% RSLogix 500 project pid_driving_pwm_analog_servo_sine_0.5-2.5ms.RSS, saved by version 8.30.00.16 %
PROJECT "UNTITLED"    % processor: Bul.1763 MicroLogix 1100 Series B %

PROGRAM FILES
  LAD 2 "CONTINUOUS"  7 rungs
  LAD 3 "DRIVESERVO"  3 rungs
  LAD 4 "PID_SCHED"  7 rungs
  LAD 5 "SINE_SIMUL"  7 rungs

DATA FILES
  O0 OUTPUT  4 elements
  I1 INPUT  6 elements
  S2 STATUS  66 elements
  B3 BINARY  1 elements
  T4 TIMER  1 elements
  C5 COUNTER  1 elements
  R6 CONTROL  1 elements
  N7 INTEGER  30 elements
  F8 FLOAT  4 elements
  L9 LONGS  8 elements
  PD10   1 elements

LADDER 2 "CONTINUOUS"
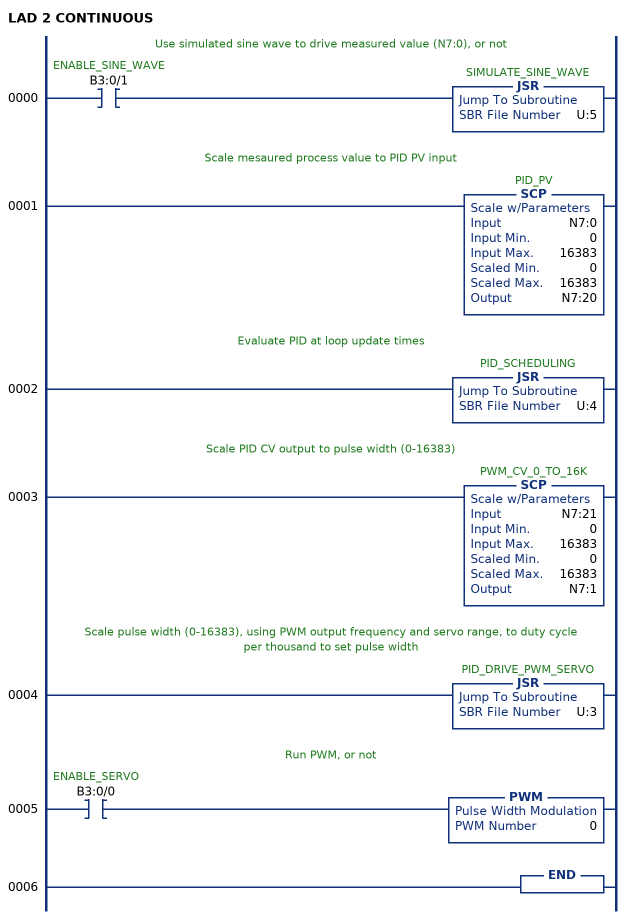
% Rung: 0 %
% Use simulated sine wave to drive measured value (N7:0), or not %
SOR XIC B3:0/1 JSR U:5 EOR
%   B3:0/1  ENABLE_SINE_WAVE %
%   U:5  SIMULATE_SINE_WAVE %
% Rung: 1 %
% Scale mesaured process value to PID PV input %
SOR SCP N7:0 0 16383 0 16383 N7:20 EOR
%   N7:0  MEASURED_VALUE %
%   N7:20  PID_PV %
% Rung: 2 %
% Evaluate PID at loop update times %
SOR JSR U:4 EOR
%   U:4  PID_SCHEDULING %
% Rung: 3 %
% Scale PID CV output to pulse width (0-16383) %
SOR SCP N7:21 0 16383 0 16383 N7:1 EOR
%   N7:21  PID_CV %
%   N7:1  PWM_CV_0_TO_16K %
% Rung: 4 %
% Scale pulse width (0-16383), using PWM output frequency and servo range, to duty cycle per thousand to set pulse width %
SOR JSR U:3 EOR
%   U:3  PID_DRIVE_PWM_SERVO %
% Rung: 5 %
% Run PWM, or not %
SOR XIC B3:0/0 PWM 0 EOR
%   B3:0/0  ENABLE_SERVO %
% Rung: 6 %
SOR END EOR

LADDER 3 "DRIVESERVO"
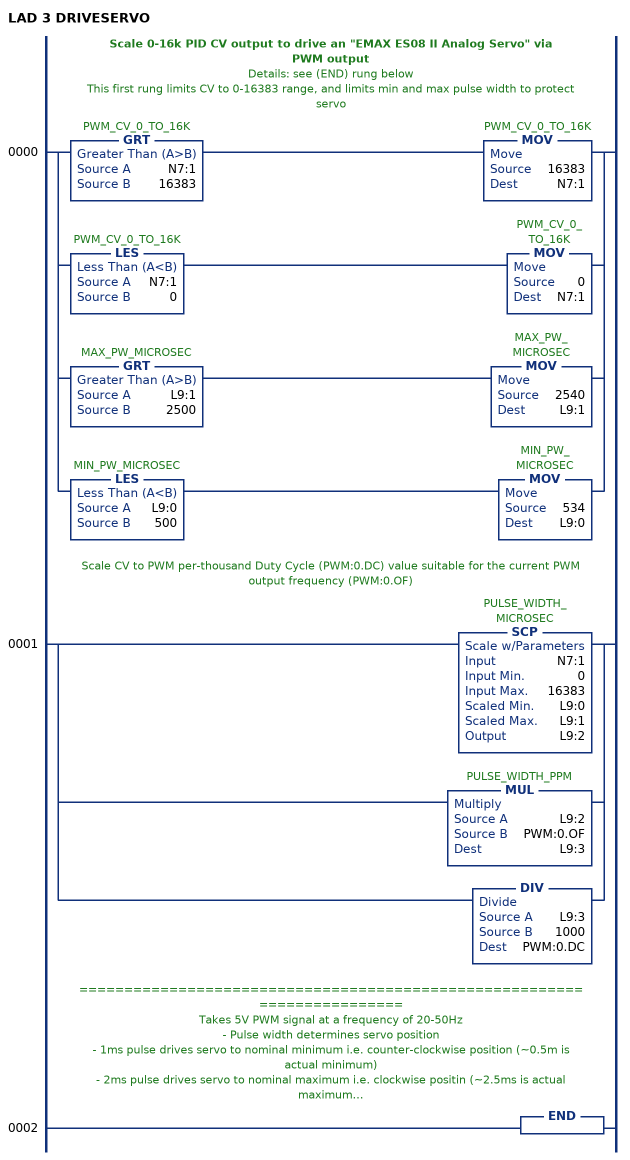
% Rung: 0 %
% TITLE: Scale 0-16k PID CV output to drive an "EMAX ES08 II Analog Servo" via PWM output %
% Details: see (END) rung below
% 
% This first rung limits CV to 0-16383 range, and limits min and max pulse width to protect servo %
SOR BST GRT N7:1 16383 MOV 16383 N7:1 NXB LES N7:1 0 MOV 0 N7:1 NXB GRT L9:1 2500 MOV 2540 L9:1 NXB LES L9:0 500 MOV 534 L9:0 BND EOR
%   N7:1  PWM_CV_0_TO_16K %
%   L9:1  MAX_PW_MICROSEC %
%   L9:0  MIN_PW_MICROSEC %
% Rung: 1 %
% Scale CV to PWM per-thousand Duty Cycle (PWM:0.DC) value suitable for the current PWM output frequency (PWM:0.OF) %
SOR BST SCP N7:1 0 16383 L9:0 L9:1 L9:2 NXB MUL L9:2 PWM:0.OF L9:3 NXB DIV L9:3 1000 PWM:0.DC BND EOR
%   N7:1  PWM_CV_0_TO_16K %
%   L9:0  MIN_PW_MICROSEC %
%   L9:1  MAX_PW_MICROSEC %
%   L9:2  PULSE_WIDTH_MICROSEC %
%   L9:3  PULSE_WIDTH_PPM %
% Rung: 2 %
% ========================================================================
% Takes 5V PWM signal at a frequency of 20-50Hz
% - Pulse width determines servo position
%   - 1ms pulse drives servo to nominal minimum i.e. counter-clockwise position (~0.5m is actual minimum)
%   - 2ms pulse drives servo to nominal maximum i.e. clockwise positin (~2.5ms is actual maximum)
% 
% PWM:0 is configured for
% - PWM:0.OUT = 2 - OUTput 2 (O:0.0/2)
% - PWM:0.OF = 100 - pulses will be generated at Output Frequency of 100Hz
% 
% PWM:0.DC (Duty Cycle) will be controlled by the program
% - .DC = 0/1000 => 0% duty cycle (always off)
% - .DC = 1000/1000 => 100% duty cycle (always on)
% - At PWM:0.OF Hz, one cycle is 1000/PWM:0.OF ms, so
%   - .DC = PWM:0.OF would generate 1ms pulses (nominal minimum postion)
%   - .DC = 2*PWM:0.OF would generate 2ms pulses (nominal maximum position)
%   - .DC = k*PWM:0.OF would generate [k]ms pulses
%   - .DC = u*PWM:0.OF/1000 would generate [u]microsecond pulses
% 
% Empirical range of Servo, PWM:0.OUT = 100Hz, 2023-04-25
% - Low:  servo is quiet at 535us pulse width (PWM0:DC=54/1000 @ 100Hz); servo hums at 534us pulse width (PWM0:DC=53/1000 @ 100Hz)
% -High:  servo is quiet at 2534us pulse width (PWM0:DC=253/1000 @ 100Hz); servo hums at 2535us pulse width (PWM0:DC=254/1000 @ 100Hz)
% ======================================================================== %
SOR END EOR

LADDER 4 "PID_SCHED"
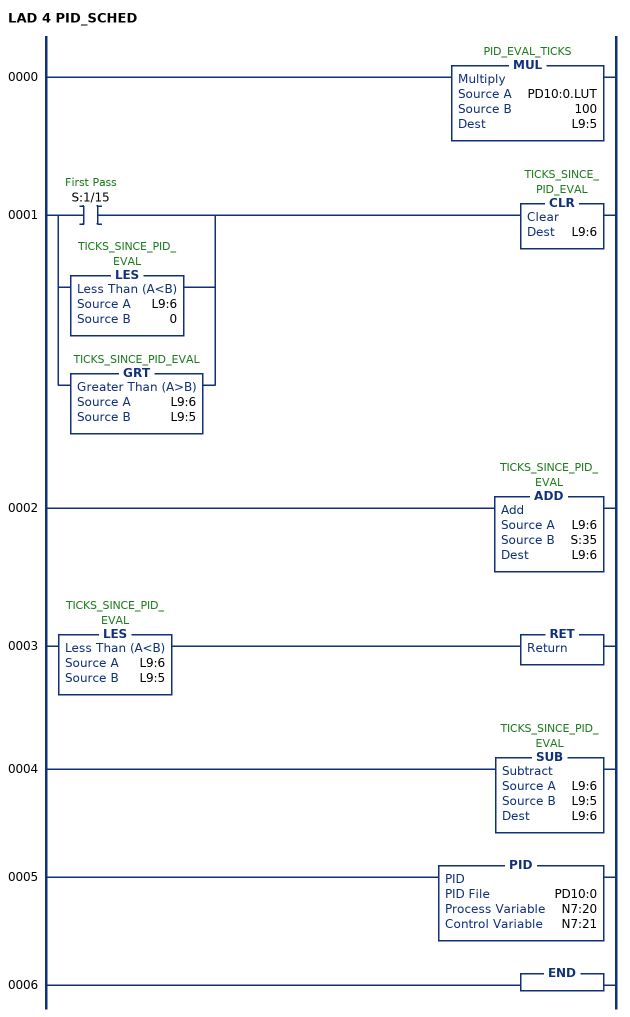
% Rung: 0 %
SOR MUL PD10:0.LUT 100 L9:5 EOR
%   L9:5  PID_EVAL_TICKS %
% Rung: 1 %
SOR BST XIC S:1/15 NXB LES L9:6 0 NXB GRT L9:6 L9:5 BND CLR L9:6 EOR
%   S:1/15  "First Pass" %
%   L9:6  TICKS_SINCE_PID_EVAL %
%   L9:5  PID_EVAL_TICKS %
% Rung: 2 %
SOR ADD L9:6 S:35 L9:6 EOR
%   L9:6  TICKS_SINCE_PID_EVAL %
%   S:35  "Last 1 ms Scan Time" %
% Rung: 3 %
SOR LES L9:6 L9:5 RET EOR
%   L9:6  TICKS_SINCE_PID_EVAL %
%   L9:5  PID_EVAL_TICKS %
% Rung: 4 %
SOR SUB L9:6 L9:5 L9:6 EOR
%   L9:6  TICKS_SINCE_PID_EVAL %
%   L9:5  PID_EVAL_TICKS %
% Rung: 5 %
SOR PID PD10:0 N7:20 N7:21 EOR
%   N7:20  PID_PV %
%   N7:21  PID_CV %
% Rung: 6 %
SOR END EOR

LADDER 5 "SINE_SIMUL"
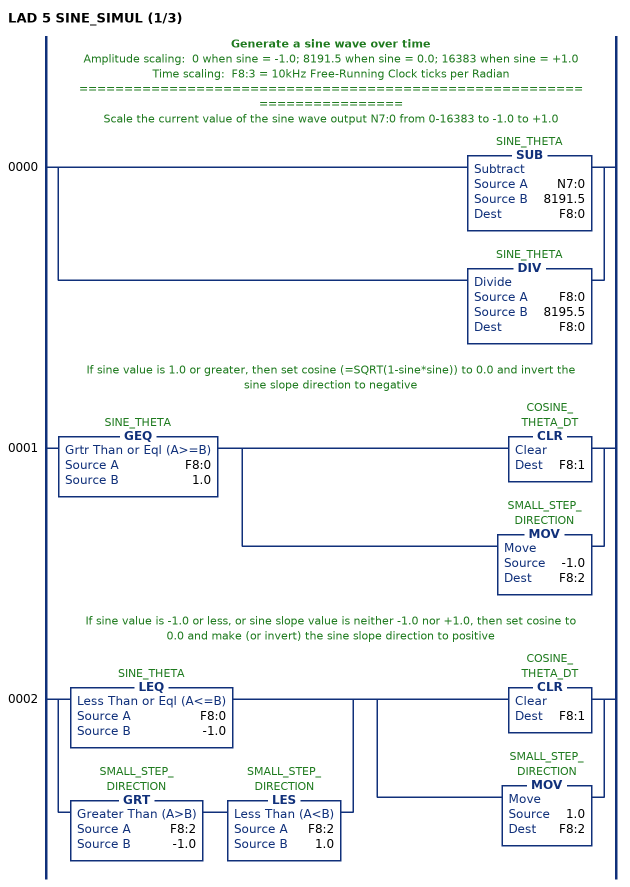
% Rung: 0 %
% TITLE: Generate a sine wave over time %
% Amplitude scaling:  0 when sine = -1.0; 8191.5 when sine = 0.0; 16383 when sine = +1.0
% Time scaling:  F8:3 = 10kHz Free-Running Clock ticks per Radian
% 
% ========================================================================
% 
% Scale the current value of the sine wave output N7:0 from 0-16383 to -1.0 to +1.0 %
SOR BST SUB N7:0 8191.5 F8:0 NXB DIV F8:0 8195.5 F8:0 BND EOR
%   N7:0  MEASURED_VALUE %
%   F8:0  SINE_THETA %
% Rung: 1 %
% If sine value is 1.0 or greater, then set cosine (=SQRT(1-sine*sine)) to 0.0 and invert the sine slope direction to negative %
SOR GEQ F8:0 1.0 BST CLR F8:1 NXB MOV -1.0 F8:2 BND EOR
%   F8:0  SINE_THETA %
%   F8:1  COSINE_THETA_DT %
%   F8:2  SMALL_STEP_DIRECTION %
% Rung: 2 %
% If sine value is -1.0 or less, or sine slope value is neither -1.0 nor +1.0, then set cosine to 0.0 and make (or invert) the sine slope direction to positive %
SOR BST LEQ F8:0 -1.0 NXB GRT F8:2 -1.0 LES F8:2 1.0 BND BST CLR F8:1 NXB MOV 1.0 F8:2 BND EOR
%   F8:0  SINE_THETA %
%   F8:2  SMALL_STEP_DIRECTION %
%   F8:1  COSINE_THETA_DT %

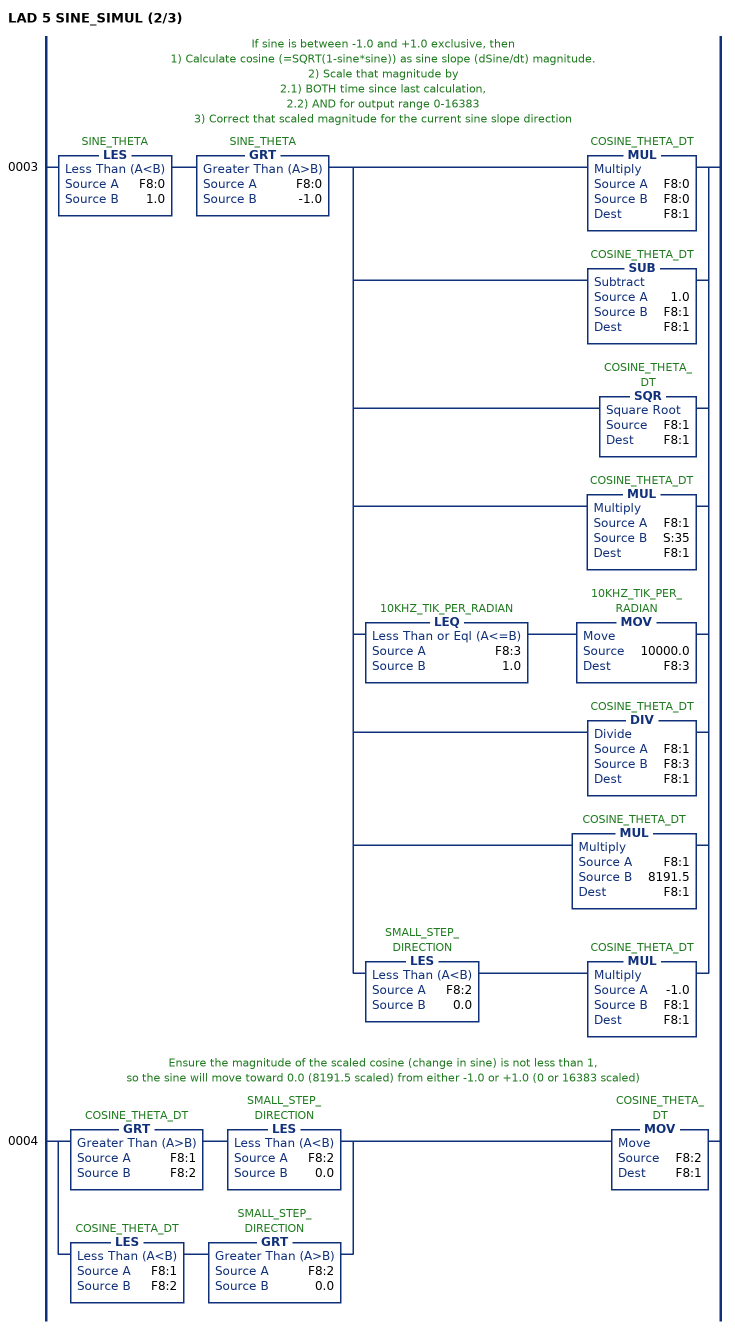
% Rung: 3 %
% If sine is between -1.0 and +1.0 exclusive, then
% 1) Calculate cosine (=SQRT(1-sine*sine)) as sine slope (dSine/dt) magnitude.
% 2) Scale that magnitude by
% 2.1) BOTH time since last calculation,
% 2.2) AND for output range 0-16383
% 3) Correct that scaled magnitude for the current sine slope direction %
SOR LES F8:0 1.0 GRT F8:0 -1.0 BST MUL F8:0 F8:0 F8:1 NXB SUB 1.0 F8:1 F8:1 NXB SQR F8:1 F8:1 NXB MUL F8:1 S:35 F8:1 NXB LEQ F8:3 1.0 MOV 10000.0 F8:3 NXB DIV F8:1 F8:3 F8:1 NXB MUL F8:1 8191.5 F8:1 NXB LES F8:2 0.0 MUL -1.0 F8:1 F8:1 BND EOR
%   F8:0  SINE_THETA %
%   F8:1  COSINE_THETA_DT %
%   S:35  "Last 1 ms Scan Time" %
%   F8:3  10KHZ_TIK_PER_RADIAN %
%   F8:2  SMALL_STEP_DIRECTION %
% Rung: 4 %
% Ensure the magnitude of the scaled cosine (change in sine) is not less than 1,
% so the sine will move toward 0.0 (8191.5 scaled) from either -1.0 or +1.0 (0 or 16383 scaled) %
SOR BST GRT F8:1 F8:2 LES F8:2 0.0 NXB LES F8:1 F8:2 GRT F8:2 0.0 BND MOV F8:2 F8:1 EOR
%   F8:1  COSINE_THETA_DT %
%   F8:2  SMALL_STEP_DIRECTION %

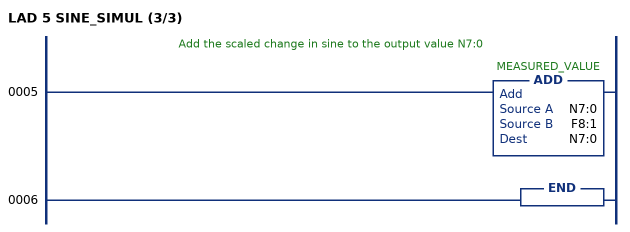
% Rung: 5 %
% Add the scaled change in sine to the output value N7:0 %
SOR ADD N7:0 F8:1 N7:0 EOR
%   N7:0  MEASURED_VALUE %
%   F8:1  COSINE_THETA_DT %
% Rung: 6 %
SOR END EOR

OTHER DOCUMENTED ADDRESSES
  N7:2  PULSE_WIDTH_MILLISEC
  PWM:0.3  OUTPUT_FREQUENCY
  PWM:0.5  DUTY_CYCLE_PER_1000

COMMENTS NOT ATTACHED TO A CURRENT RUNG
  B3:3/1: Turn on the LED for any B that is stopped
  B3:1/0: Keep track of whether any B will be turned on during this scan
  B3:3/3: If any B-stop button is pressed when that B is on, the light that B's LED, and leave it on until any B is started
  B3:0/3: If a B-start button is pressed while no B-LEDs are lit, then turn on that B
    If any B has been stopped above during this scan, then a B-LED will be lit, use that to turn off all Bs
  B3:1: Clear any start or stop buttons
  B3:3/5: If any B is stopped, then turn on that LED and leave it on until any start button is pressed
  B3:0/5: If any start button is pressed, then turn on that B and leave it on, until any B is stopped and an LED is turned on on the rung above

DATA TABLE (non-zero values as saved)
DATA C5
% .PRE .ACC %
% C5:0 % 50 0
DATA F8
% F8:0 % 0 0 0 10000
DATA L9
% L9:0 % 500 2500 0 0 0
